// TIA Portal V18 export
FUNCTION_BLOCK "LGasp_Ansa4livelli"   // FB20109, LAD
TITLE = Gestione ansa con 3 laser da IOLink
{ S7_Optimized_Access := 'TRUE' }
VERSION : 0.1
// stored: AutoNumber false, IsIECCheckEnabled false, IsRetainMemResEnabled false, MemoryReserve 100, SetENOAutomatically false, UDAEnableTagReadback false
   VAR_INPUT
      i_Laser1 { ExternalAccessible := 'False'; ExternalVisible := 'False'; ExternalWritable := 'False'} : Int;   // Laser collegato in IOLink
      i_Laser2 { ExternalAccessible := 'False'; ExternalVisible := 'False'; ExternalWritable := 'False'} : Int;   // Laser collegato in IOLink
      i_Laser3 { ExternalAccessible := 'False'; ExternalVisible := 'False'; ExternalWritable := 'False'} : Int;   // Laser collegato in IOLink
      i_abilitaLaser2 { ExternalAccessible := 'False'; ExternalVisible := 'False'; ExternalWritable := 'False'} : Bool;   // 1=Abilita laser
      i_abilitaLaser3 { ExternalAccessible := 'False'; ExternalVisible := 'False'; ExternalWritable := 'False'} : Bool;   // 1=Abilita laser
      i_AutoSTZsuccessivaAnsa { ExternalAccessible := 'False'; ExternalVisible := 'False'; ExternalWritable := 'False'} : Bool;   // Automatico stazione dopo l'ansa
      i_AvantiLamiera { ExternalAccessible := 'False'; ExternalVisible := 'False'; ExternalWritable := 'False'} : Bool;   // Lamiera in movimento avanti per jog profila/marcia semiautomatica o marcia automatica
      i_FTCfineLamiera { ExternalAccessible := 'False'; ExternalVisible := 'False'; ExternalWritable := 'False'} : Bool;   // fotocellula fine lamiera prima dell'ansa
      i_Reset { ExternalAccessible := 'False'; ExternalVisible := 'False'; ExternalWritable := 'False'} : Bool;
      i_SensoreTavola { ExternalAccessible := 'False'; ExternalVisible := 'False'; ExternalWritable := 'False'} : Bool;   // sensore tavola accompagnamento
      i_DS_AnsaBassa { ExternalAccessible := 'False'; ExternalVisible := 'False'; ExternalWritable := 'False'} : LReal;
      i_DS_AnsaMedioBassa { ExternalAccessible := 'False'; ExternalVisible := 'False'; ExternalWritable := 'False'} : LReal;
      i_DS_AnsaMedioAlta { ExternalAccessible := 'False'; ExternalVisible := 'False'; ExternalWritable := 'False'} : LReal;
      i_DS_AnsaAlta { ExternalAccessible := 'False'; ExternalVisible := 'False'; ExternalWritable := 'False'} : LReal;
   END_VAR
   VAR_OUTPUT
      o_ansa { ExternalAccessible := 'False'; ExternalVisible := 'False'; ExternalWritable := 'False'} : "LGasp_typeAnsa4Livelli";
      o_FLT_AnsaAlta { ExternalAccessible := 'False'; ExternalVisible := 'False'; ExternalWritable := 'False'} : Bool;
      o_FLT_PosizioneTavola { ExternalAccessible := 'False'; ExternalVisible := 'False'; ExternalWritable := 'False'} : Bool;
      o_FLT_ValoreLaser { ExternalAccessible := 'False'; ExternalVisible := 'False'; ExternalWritable := 'False'} : Bool;
   END_VAR
   VAR
      s_MediaValoriL1 { ExternalAccessible := 'False'; ExternalVisible := 'False'; ExternalWritable := 'False'} : DInt;
      s_MediaValoriL2 { ExternalAccessible := 'False'; ExternalVisible := 'False'; ExternalWritable := 'False'} : DInt;
      s_MediaValoriL3 { ExternalAccessible := 'False'; ExternalVisible := 'False'; ExternalWritable := 'False'} : DInt;
      s_sommaL1 { ExternalAccessible := 'False'; ExternalVisible := 'False'; ExternalWritable := 'False'} : DInt;
      s_sommaL2 { ExternalAccessible := 'False'; ExternalVisible := 'False'; ExternalWritable := 'False'} : DInt;
      s_sommaL3 { ExternalAccessible := 'False'; ExternalVisible := 'False'; ExternalWritable := 'False'} : DInt;
      s_PuntatoreL1 { ExternalAccessible := 'False'; ExternalVisible := 'False'; ExternalWritable := 'False'} : DInt;
      s_PuntatoreL2 { ExternalAccessible := 'False'; ExternalVisible := 'False'; ExternalWritable := 'False'} : DInt;
      s_PuntatoreL3 { ExternalAccessible := 'False'; ExternalVisible := 'False'; ExternalWritable := 'False'} : DInt;
      s_ValoreLaser : DInt;
      s_ValoreAnsa { ExternalAccessible := 'False'; ExternalVisible := 'False'; ExternalWritable := 'False'} : LReal;
      s_consenso_da_ansa { ExternalAccessible := 'False'; ExternalVisible := 'False'; ExternalWritable := 'False'} : Bool;
   END_VAR
   VAR RETAIN
      s_DM { ExternalAccessible := 'False'; ExternalVisible := 'False'; ExternalWritable := 'False'} : Struct
         filtroMinAnsa { ExternalAccessible := 'False'; ExternalVisible := 'False'; ExternalWritable := 'False'} : Time := t#100ms;   // filtro su allarme minima ansa
         filtroLaserFLT { ExternalAccessible := 'False'; ExternalVisible := 'False'; ExternalWritable := 'False'} : Time := t#1s;   // filtro su errore lettura laser
         ValoriMedia { ExternalAccessible := 'False'; ExternalVisible := 'False'; ExternalWritable := 'False'} : DInt := 10;
         SogliaMinima { ExternalAccessible := 'False'; ExternalVisible := 'False'; ExternalWritable := 'False'} : Int := 100;
         SogliaMassima { ExternalAccessible := 'False'; ExternalVisible := 'False'; ExternalWritable := 'False'} : Int := 4900;
      END_STRUCT;
   END_VAR
   VAR
      IEC_Timer_FaultLaser { ExternalAccessible := 'False'; ExternalVisible := 'False'; ExternalWritable := 'False'} : TON_TIME;
      IEC_Timer_FaultAnsaAlta { ExternalAccessible := 'False'; ExternalVisible := 'False'; ExternalWritable := 'False'} : TON_TIME;
   END_VAR
   VAR_TEMP   // added for the SCL form of the ladder/FBD networks
      _w1 : Bool;
      _w2 : Bool;
      _w3 : Bool;
   END_VAR
BEGIN

REGION Network 1 (SCL): INFORMAZIONI GENERALI
   //================================================================================
   // Gasparini Spa
   //--------------------------------------------------------------------------------
   // Libreria: LGasp_V17 
   // Funzionalità: Gestione ansa gestita da massimo 3 laser 
   // Commessa in cui è stata testata: Micron 303/304
   // Programmatore di riferimento per test: XXXXXX
   //--------------------------------------------------------------------------------
   // Change log table:
   // Versione Data        Autore          Modifiche
   // 01.00.00 08.04.2021  Lcg          Rilascio funzione
   // 02.00.00 01.08.2021  Lcg         Migrazione a TIA 17
   // 02.00.01 09.06.2022  Lcg         Aggiunti due timer, il primo filtra il segnale del laser, il secondo permette di ritardare l'allarme minima ansa.
   // 02.00.02 20.06.2022  Lcg         Modificato allarme minima ansa in modo intervenga anche in manuale , inseriti i valori dei timer come DM
   // 02.00.03 23.12.2022  Lcg         Aggiunto segnale di avanti materiale nella generazione dell'allarme di minima ansa. Questo permette di resettare 
   //                                  l'allarme minima ansa e riempire l'ansa nuovamente.
   //                                  Messi i valori delle costanti sotto la struttura DM per poterli modificare senza aprire la libreria.
   // 03.00.00 06.02.2023  Lcg         Migrazione a TIA 18
   //--------------------------------------------------------------------------------
   // Nota: 
   //
   //================================================================================
END_REGION

REGION Network 2: Somma letture + incrementa puntatore
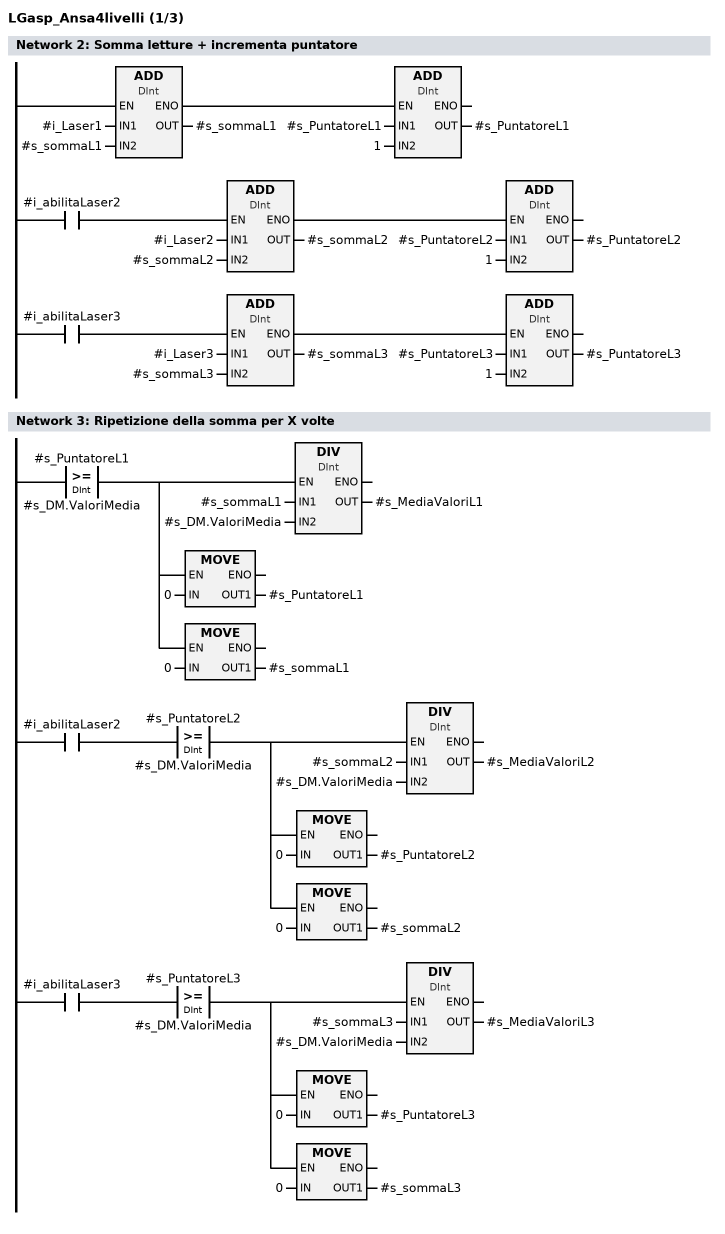
   RUNG wire#powerrail
      { S7_Templates := "SrcType := DInt"; S7_GenerateENO := "TRUE" } Add(in1 := #i_Laser1, in2 := #s_sommaL1, out => #s_sommaL1)
      { S7_Templates := "SrcType := DInt"; S7_GenerateENO := "TRUE" } Add(in1 := #s_PuntatoreL1, in2 := 1, out => #s_PuntatoreL1)
   END_RUNG
   RUNG wire#powerrail
      Contact( #i_abilitaLaser2 )
      { S7_Templates := "SrcType := DInt"; S7_GenerateENO := "TRUE" } Add(in1 := #i_Laser2, in2 := #s_sommaL2, out => #s_sommaL2)
      { S7_Templates := "SrcType := DInt"; S7_GenerateENO := "TRUE" } Add(in1 := #s_PuntatoreL2, in2 := 1, out => #s_PuntatoreL2)
   END_RUNG
   RUNG wire#powerrail
      Contact( #i_abilitaLaser3 )
      { S7_Templates := "SrcType := DInt"; S7_GenerateENO := "TRUE" } Add(in1 := #i_Laser3, in2 := #s_sommaL3, out => #s_sommaL3)
      { S7_Templates := "SrcType := DInt"; S7_GenerateENO := "TRUE" } Add(in1 := #s_PuntatoreL3, in2 := 1, out => #s_PuntatoreL3)
   END_RUNG
   // the same network as SCL:
   // ENO of a box is taken as its EN; it also drops when the box reports an error
   #s_sommaL1 := #i_Laser1 + #s_sommaL1;
   #s_PuntatoreL1 := #s_PuntatoreL1 + 1;
   IF #i_abilitaLaser2 THEN
       #s_sommaL2 := #i_Laser2 + #s_sommaL2;
       #s_PuntatoreL2 := #s_PuntatoreL2 + 1;
   END_IF;
   IF #i_abilitaLaser3 THEN
       #s_sommaL3 := #i_Laser3 + #s_sommaL3;
       #s_PuntatoreL3 := #s_PuntatoreL3 + 1;
   END_IF;
END_REGION

REGION Network 3: Ripetizione della somma per X volte
   RUNG wire#powerrail
      { S7_Templates := "SrcType := DInt" } GE_Contact(in1 := #s_PuntatoreL1, in2 := #s_DM.ValoriMedia)
      wire#w1
      { S7_Templates := "SrcType := DInt"; S7_GenerateENO := "TRUE" } Div(in1 := #s_sommaL1, in2 := #s_DM.ValoriMedia, out => #s_MediaValoriL1)
   END_RUNG
   RUNG wire#w1
      Move(in := 0, out1 => #s_PuntatoreL1)
   END_RUNG
   RUNG wire#w1
      Move(in := 0, out1 => #s_sommaL1)
   END_RUNG
   RUNG wire#powerrail
      Contact( #i_abilitaLaser2 )
      { S7_Templates := "SrcType := DInt" } GE_Contact(in1 := #s_PuntatoreL2, in2 := #s_DM.ValoriMedia)
      wire#w2
      { S7_Templates := "SrcType := DInt"; S7_GenerateENO := "TRUE" } Div(in1 := #s_sommaL2, in2 := #s_DM.ValoriMedia, out => #s_MediaValoriL2)
   END_RUNG
   RUNG wire#w2
      Move(in := 0, out1 => #s_PuntatoreL2)
   END_RUNG
   RUNG wire#w2
      Move(in := 0, out1 => #s_sommaL2)
   END_RUNG
   RUNG wire#powerrail
      Contact( #i_abilitaLaser3 )
      { S7_Templates := "SrcType := DInt" } GE_Contact(in1 := #s_PuntatoreL3, in2 := #s_DM.ValoriMedia)
      wire#w3
      { S7_Templates := "SrcType := DInt"; S7_GenerateENO := "TRUE" } Div(in1 := #s_sommaL3, in2 := #s_DM.ValoriMedia, out => #s_MediaValoriL3)
   END_RUNG
   RUNG wire#w3
      Move(in := 0, out1 => #s_PuntatoreL3)
   END_RUNG
   RUNG wire#w3
      Move(in := 0, out1 => #s_sommaL3)
   END_RUNG
   // the same network as SCL:
   IF #s_PuntatoreL1 >= #s_DM.ValoriMedia THEN #s_MediaValoriL1 := #s_sommaL1 / #s_DM.ValoriMedia; END_IF;
   #_w1 := #s_PuntatoreL1 >= #s_DM.ValoriMedia;
   IF #_w1 THEN
       #s_PuntatoreL1 := 0;
       #s_sommaL1 := 0;
   END_IF;
   IF #i_abilitaLaser2 AND (#s_PuntatoreL2 >= #s_DM.ValoriMedia) THEN
       #s_MediaValoriL2 := #s_sommaL2 / #s_DM.ValoriMedia;
   END_IF;
   #_w2 := #i_abilitaLaser2 AND (#s_PuntatoreL2 >= #s_DM.ValoriMedia);
   IF #_w2 THEN
       #s_PuntatoreL2 := 0;
       #s_sommaL2 := 0;
   END_IF;
   IF #i_abilitaLaser3 AND (#s_PuntatoreL3 >= #s_DM.ValoriMedia) THEN
       #s_MediaValoriL3 := #s_sommaL3 / #s_DM.ValoriMedia;
   END_IF;
   #_w3 := #i_abilitaLaser3 AND (#s_PuntatoreL3 >= #s_DM.ValoriMedia);
   IF #_w3 THEN
       #s_PuntatoreL3 := 0;
       #s_sommaL3 := 0;
   END_IF;
END_REGION

REGION Network 4: Viene preso il valore laser più basso
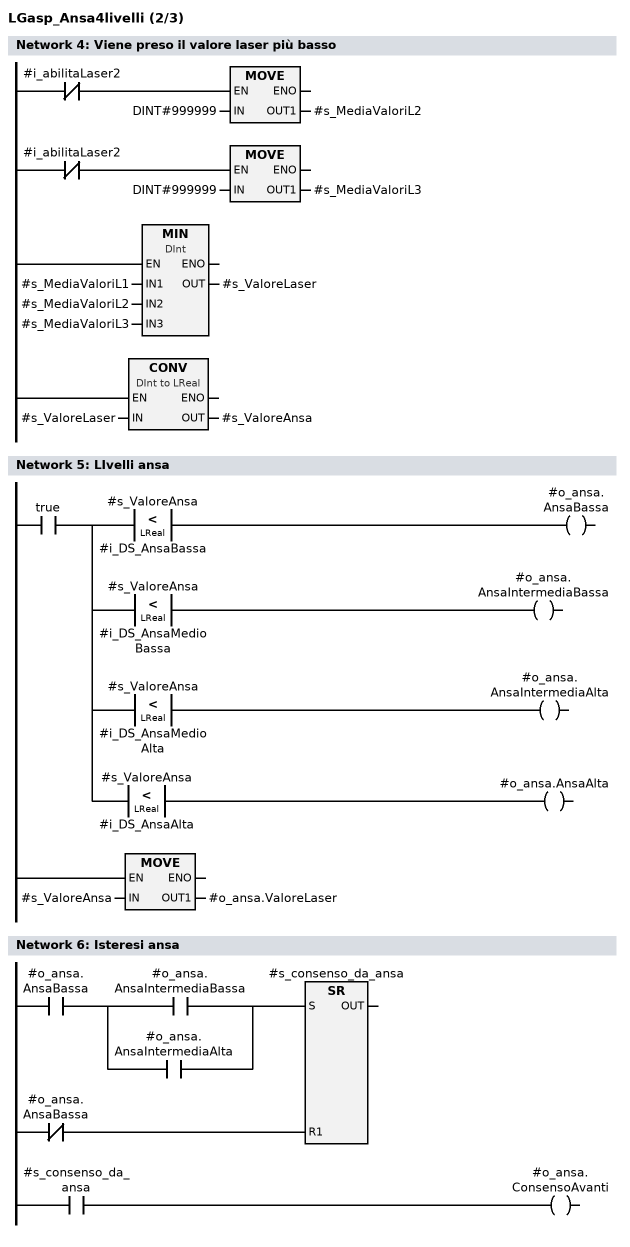
   RUNG wire#powerrail
      I_Contact( #i_abilitaLaser2 )
      Move(in := DINT#999999, out1 => #s_MediaValoriL2)
   END_RUNG
   RUNG wire#powerrail
      I_Contact( #i_abilitaLaser2 )
      Move(in := DINT#999999, out1 => #s_MediaValoriL3)
   END_RUNG
   RUNG wire#powerrail
      { S7_Templates := "[card := 3, value_type := DInt]" } MIN(in1 := #s_MediaValoriL1, in2 := #s_MediaValoriL2, in3 := #s_MediaValoriL3, out => #s_ValoreLaser)
   END_RUNG
   RUNG wire#powerrail
      { S7_Templates := "[SrcType := DInt, DestType := LReal]" } Convert(in := #s_ValoreLaser, out => #s_ValoreAnsa)
   END_RUNG
   // the same network as SCL:
   IF NOT #i_abilitaLaser2 THEN
       #s_MediaValoriL2 := DINT#999999;
       #s_MediaValoriL3 := DINT#999999;
   END_IF;
   #s_ValoreLaser := MIN(IN1 := #s_MediaValoriL1, IN2 := #s_MediaValoriL2, IN3 := #s_MediaValoriL3);
   #s_ValoreAnsa := DINT_TO_LREAL(#s_ValoreLaser);
END_REGION

REGION Network 5: LIvelli ansa
   RUNG wire#powerrail
      Contact( true )
      wire#w1
      { S7_Templates := "SrcType := LReal" } LT_Contact(in1 := #s_ValoreAnsa, in2 := #i_DS_AnsaBassa)
      Coil( #o_ansa.AnsaBassa )
   END_RUNG
   RUNG wire#w1
      { S7_Templates := "SrcType := LReal" } LT_Contact(in1 := #s_ValoreAnsa, in2 := #i_DS_AnsaMedioBassa)
      Coil( #o_ansa.AnsaIntermediaBassa )
   END_RUNG
   RUNG wire#w1
      { S7_Templates := "SrcType := LReal" } LT_Contact(in1 := #s_ValoreAnsa, in2 := #i_DS_AnsaMedioAlta)
      Coil( #o_ansa.AnsaIntermediaAlta )
   END_RUNG
   RUNG wire#w1
      { S7_Templates := "SrcType := LReal" } LT_Contact(in1 := #s_ValoreAnsa, in2 := #i_DS_AnsaAlta)
      Coil( #o_ansa.AnsaAlta )
   END_RUNG
   RUNG wire#powerrail
      Move(in := #s_ValoreAnsa, out1 => #o_ansa.ValoreLaser)
   END_RUNG
   // the same network as SCL:
   #o_ansa.AnsaBassa := true AND (#s_ValoreAnsa < #i_DS_AnsaBassa);
   #o_ansa.AnsaIntermediaBassa := true AND (#s_ValoreAnsa < #i_DS_AnsaMedioBassa);
   #o_ansa.AnsaIntermediaAlta := true AND (#s_ValoreAnsa < #i_DS_AnsaMedioAlta);
   #o_ansa.AnsaAlta := true AND (#s_ValoreAnsa < #i_DS_AnsaAlta);
   #o_ansa.ValoreLaser := #s_ValoreAnsa;
END_REGION

REGION Network 6: Isteresi ansa
   RUNG wire#powerrail
      Contact( #o_ansa.AnsaBassa )
      wire#w1
      Contact( #o_ansa.AnsaIntermediaBassa )
      wire#w2
      S_SR(operand := #s_consenso_da_ansa, r1 := wire#w3)
   END_RUNG
   RUNG wire#w1
      Contact( #o_ansa.AnsaIntermediaAlta )
   END_RUNG wire#w2
   RUNG wire#powerrail
      I_Contact( #o_ansa.AnsaBassa )
   END_RUNG wire#w3
   RUNG wire#powerrail
      Contact( #s_consenso_da_ansa )
      Coil( #o_ansa.ConsensoAvanti )
   END_RUNG
   // the same network as SCL:
   IF #o_ansa.AnsaBassa AND (#o_ansa.AnsaIntermediaBassa OR #o_ansa.AnsaIntermediaAlta) THEN
       #s_consenso_da_ansa := TRUE;   // SR flip-flop
   END_IF;
   IF NOT #o_ansa.AnsaBassa THEN #s_consenso_da_ansa := FALSE; END_IF;
   #o_ansa.ConsensoAvanti := #s_consenso_da_ansa;
END_REGION

REGION Network 7: Allarmi ansa
   // Aggiunti due timer, il primo filtra il segnale del laser, il secondo permette di ritardare l'allarme quando si ridà la marcia impianto
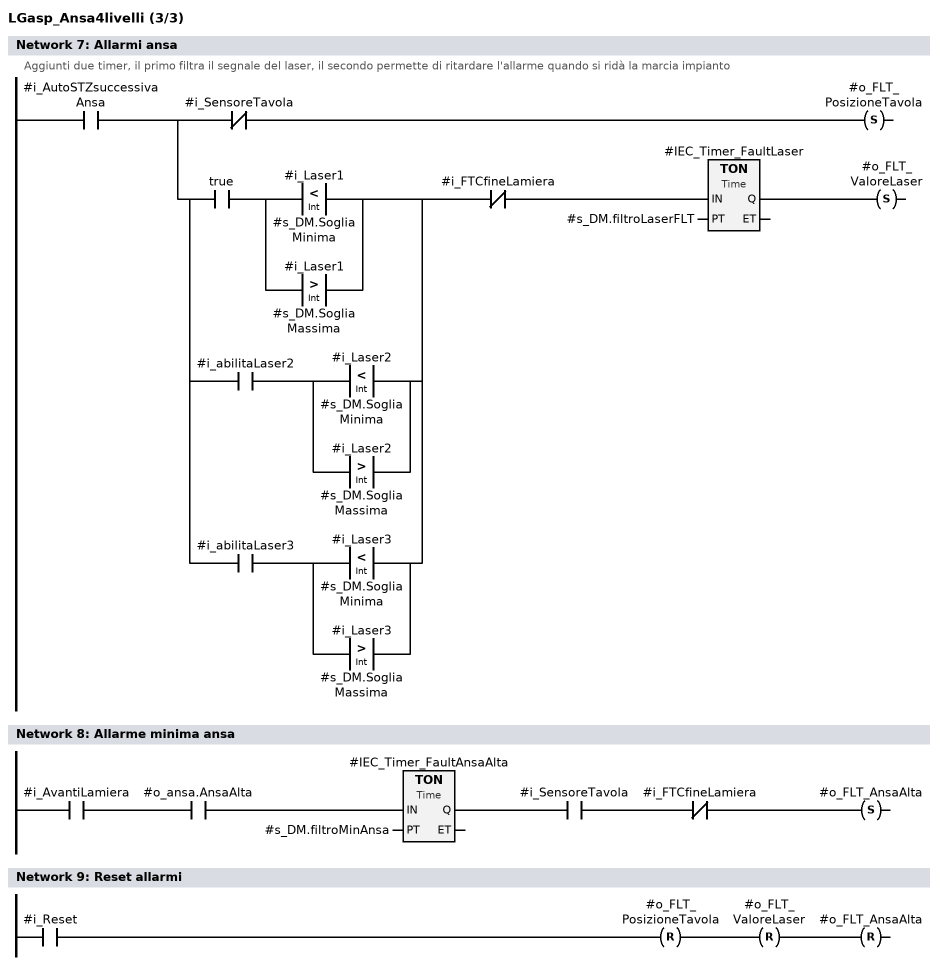
   RUNG wire#powerrail
      Contact( #i_AutoSTZsuccessivaAnsa )
      wire#w1
      I_Contact( #i_SensoreTavola )
      S_Coil( #o_FLT_PosizioneTavola )
   END_RUNG
   RUNG wire#w1
      Contact( true )
      wire#w2
      { S7_Templates := "SrcType := Int" } LT_Contact(in1 := #i_Laser1, in2 := #s_DM.SogliaMinima)
      wire#w3
      I_Contact( #i_FTCfineLamiera )
      { S7_Templates := "time_type := Time" } #IEC_Timer_FaultLaser.TON(pt := #s_DM.filtroLaserFLT, et =>)
      S_Coil( #o_FLT_ValoreLaser )
   END_RUNG
   RUNG wire#w2
      { S7_Templates := "SrcType := Int" } GT_Contact(in1 := #i_Laser1, in2 := #s_DM.SogliaMassima)
   END_RUNG wire#w3
   RUNG wire#w1
      Contact( #i_abilitaLaser2 )
      wire#w4
      { S7_Templates := "SrcType := Int" } LT_Contact(in1 := #i_Laser2, in2 := #s_DM.SogliaMinima)
   END_RUNG wire#w3
   RUNG wire#w4
      { S7_Templates := "SrcType := Int" } GT_Contact(in1 := #i_Laser2, in2 := #s_DM.SogliaMassima)
   END_RUNG wire#w3
   RUNG wire#w1
      Contact( #i_abilitaLaser3 )
      wire#w5
      { S7_Templates := "SrcType := Int" } LT_Contact(in1 := #i_Laser3, in2 := #s_DM.SogliaMinima)
   END_RUNG wire#w3
   RUNG wire#w5
      { S7_Templates := "SrcType := Int" } GT_Contact(in1 := #i_Laser3, in2 := #s_DM.SogliaMassima)
   END_RUNG wire#w3
   // the same network as SCL:
   IF #i_AutoSTZsuccessivaAnsa AND NOT #i_SensoreTavola THEN #o_FLT_PosizioneTavola := TRUE; END_IF;
   #IEC_Timer_FaultLaser(IN := #i_AutoSTZsuccessivaAnsa AND ((true AND ((#i_Laser1 < #s_DM.SogliaMinima) OR (#i_Laser1 > #s_DM.SogliaMassima))) OR (#i_abilitaLaser2 AND ((#i_Laser2 < #s_DM.SogliaMinima) OR (#i_Laser2 > #s_DM.SogliaMassima))) OR (#i_abilitaLaser3 AND ((#i_Laser3 < #s_DM.SogliaMinima) OR (#i_Laser3 > #s_DM.SogliaMassima)))) AND NOT #i_FTCfineLamiera,   // TON
                         PT := #s_DM.filtroLaserFLT);
   IF #IEC_Timer_FaultLaser.Q THEN #o_FLT_ValoreLaser := TRUE; END_IF;
END_REGION

REGION Network 8: Allarme minima ansa
   RUNG wire#powerrail
      Contact( #i_AvantiLamiera )
      Contact( #o_ansa.AnsaAlta )
      { S7_Templates := "time_type := Time" } #IEC_Timer_FaultAnsaAlta.TON(pt := #s_DM.filtroMinAnsa, et =>)
      Contact( #i_SensoreTavola )
      I_Contact( #i_FTCfineLamiera )
      S_Coil( #o_FLT_AnsaAlta )
   END_RUNG
   // the same network as SCL:
   #IEC_Timer_FaultAnsaAlta(IN := #i_AvantiLamiera AND #o_ansa.AnsaAlta, PT := #s_DM.filtroMinAnsa);   // TON
   IF #IEC_Timer_FaultAnsaAlta.Q AND #i_SensoreTavola AND NOT #i_FTCfineLamiera THEN
       #o_FLT_AnsaAlta := TRUE;
   END_IF;
END_REGION

REGION Network 9: Reset allarmi
   RUNG wire#powerrail
      Contact( #i_Reset )
      R_Coil( #o_FLT_PosizioneTavola )
      R_Coil( #o_FLT_ValoreLaser )
      R_Coil( #o_FLT_AnsaAlta )
   END_RUNG
   // the same network as SCL:
   IF #i_Reset THEN
       #o_FLT_PosizioneTavola := FALSE;
       #o_FLT_ValoreLaser := FALSE;
       #o_FLT_AnsaAlta := FALSE;
   END_IF;
END_REGION
END_FUNCTION_BLOCK
